(*~
		<docu>
			<summary>
				Default implementation of DAQ.	
				<note type="tip">
					 This type is partially extended by IVF to retrieve data from the DAQ in IVF application.			
				</note>												 
			</summary>		
			<code>
			   // Intializes DAQ retrieval into applications logger
				..._daq.StartDaq();
			</code>
			<code>
				FUNCTION_BLOCK DaqUsage EXTENDS TcoCore.TcoObject
				VAR
					_daq : TcoCore.TcoDaq(THIS^);
					_counter : INT;
                    _myData : MyDataStruct;
				END_VAR
				//---------------------------------------------
				_counter := _counter + 1;
			    _daq.PushData(ADR(_myData), SIZEOF(MyDataStruct));
			</code>		
		</docu>
~*)
FUNCTION_BLOCK TcoDaq EXTENDS TcoObject IMPLEMENTS ITcoDaq
VAR
	 (*~
		<docu>
			<summary>
				Circural buffer for this DAQ.					 
			</summary>				
		</docu>
    ~*)
	_buffer : TcoDaqItem;

	(*~
		<docu>
			<summary>
				Circular carret of of the DAQ buffer. 					 
			</summary>				
		</docu>
    ~*)
	_plcCarret : INT;
END_VAR

VAR CONSTANT
	(*~
		<docu>
			<summary>
				Max number of buffered DAQ entries in bytes. 				 
			</summary>				
		</docu>
    ~*)
	MAX_DAQ_BUFFER_INDEX : INT := 5000;
    
	(*~
		<docu>
			<summary>
				Max number of buffered DAQ entries in bytes before set a dequeuing request. 				 
			</summary>				
		</docu>
    ~*)
	MAX_DAQ_BYTE_LENGHT : INT := 500; 

END_VAR

(*~
		<docu>
			<summary>
				Pushes the data to DAQ buffer.
				See also `PushData`
				<note type="important">When using this method in a cyclical environment the data will be push each time it is called. You may easily overrun the DAQ buffer.</note>				 
			</summary>				
		</docu>
~*)
METHOD PUBLIC Push
VAR_INPUT
	(*~
		<docu>
			<summary>
				Pointer on DAQ entry.				 
			</summary>				
		</docu>
	~*)
    pData : PVOID;
	(*~
		<docu>
			<summary>
				Size of DAQ entry in byte.				 
			</summary>				
		</docu>
	~*)
    DataSize : INT;
END_VAR
VAR
	_tmpDaqEntry : TcoDaqEntry;
END_VAR
IF(Parent <> 0 AND_THEN Parent.Context <> 0 AND_THEN Parent.Context.RealTimeClock <> 0) THEN
	_tmpDaqEntry.TimeStamp :=  Parent.Context.RealTimeClock.NowLocal();	
	_tmpDaqEntry.Cycle := Parent.Context.StartCycleCount;	
END_IF;	

_tmpDaqEntry.pData := pData;
_tmpDaqEntry.DataSize := DataSize;
_tmpDaqEntry.Identity := 0;
_tmpDaqEntry.MessageDigest := 0;
	

PushData(_tmpDaqEntry);
END_METHOD

(*~
		<docu>
			<summary>
				Pushes the data to DAQ buffer.
				See also `Push`
				<note:important>
						TODO: This method is typically invoked from a `TcoMessenger`. 
						TODO: Depending on settings of the messenger the messages can be logged on rising edge of the message, to prevent buffer overrun.
						TODO: For details see `TcoMessengerSettings`.
				</note>				 
			</summary>				
		</docu>
~*)
METHOD PushData
VAR_INPUT
	inDaqEntry	: TcoDaqEntry;
END_VAR
// Check enough free space  for a new DAQ entry
IF((_plcCarret + inDaqEntry.DataSize) > MAX_DAQ_BUFFER_INDEX) THEN
		_plcCarret := 1;
END_IF

IF((_plcCarret + inDaqEntry.DataSize) > MAX_DAQ_BYTE_LENGHT) THEN
		_buffer.ExpectDequeing := TRUE;
END_IF


Tc2_System.MEMCPY(
    destAddr := _buffer.Data[_plcCarret], 
    srcAddr  := inDaqEntry.pData,
    n        := TO_UDINT(inDaqEntry.DataSize)
);

_plcCarret := _plcCarret + inDaqEntry.DataSize;
END_METHOD

END_FUNCTION_BLOCK

(* stored: Version 1.1.0.1
   POU TcoDaq: Id {8fe8c386-5d63-07cd-3c39-fabdbfd58ac3}, SpecialFunc None
   Method Push: Id {25f40a70-ac72-03b6-026a-0e415c9bfaa5}
   Method PushData: Id {e0b3ca52-7de2-01ac-312e-a838125297f2} *)
